Fanuc TP program (LS listing): _bgl_override.ls

/PROG  _BGL_OVERRIDE
/ATTR
OWNER		= MNEDITOR;
COMMENT		= "";
PROG_SIZE	= 233;
CREATE		= DATE 00-01-13  TIME 01:27:18;
MODIFIED	= DATE 00-01-13  TIME 01:39:26;
FILE_NAME	= ;
VERSION		= 0;
LINE_COUNT	= 3;
MEMORY_SIZE	= 625;
PROTECT		= READ_WRITE;
TCD:  STACK_SIZE	= 0,
      TASK_PRIORITY	= 50,
      TIME_SLICE	= 0,
      BUSY_LAMP_OFF	= 0,
      ABORT_REQUEST	= 0,
      PAUSE_REQUEST	= 0;
DEFAULT_GROUP	= *,*,*,*,*;
CONTROL_CODE	= 00000000 00000000;
LOCAL_REGISTERS	= 0,0,0;
/APPL
/APPL

AUTO_SINGULARITY_HEADER;
  ENABLE_SINGULARITY_AVOIDANCE   : FALSE;
/MN
   1:  IF (!SO[7:TP enabled]) THEN ;
   2:  $mcr.$genoverride=100 ;
   3:  ENDIF ;
/POS
/END
